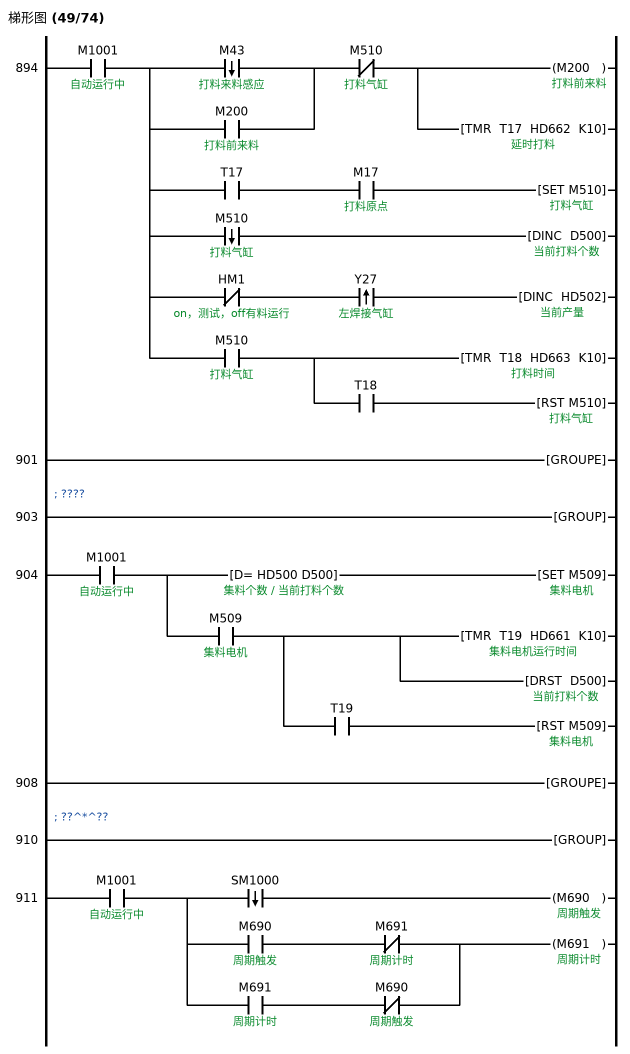
[picture p48: 梯形图 rows 894-911]
LD     M1001	; 自动运行中
MPS
LDF    M43	; 打料来料感应
OR     M200	; 打料前来料
ANB
ANI    M510	; 打料气缸
OUT    M200	; 打料前来料
TMR    T17 HD662 K10	; 延时打料
MRD
AND    T17
AND    M17	; 打料原点
SET    M510	; 打料气缸
MRD
ANDF   M510	; 打料气缸
DINC   D500	; 当前打料个数
MRD
ANI    HM1	; on，测试，off有料运行
ANDP   Y27	; 左焊接气缸
DINC   HD502	; 当前产量
MPP
AND    M510	; 打料气缸
TMR    T18 HD663 K10	; 打料时间
AND    T18
RST    M510	; 打料气缸
GROUPE
; ????
GROUP
LD     M1001	; 自动运行中
MPS
DAND=  HD500 D500	; 集料个数 / 当前打料个数
SET    M509	; 集料电机
MPP
AND    M509	; 集料电机
TMR    T19 HD661 K10	; 集料电机运行时间
DRST   D500	; 当前打料个数
AND    T19
RST    M509	; 集料电机
GROUPE
; ??^*^??
GROUP
LD     M1001	; 自动运行中
MPS
ANDF   SM1000
OUT    M690	; 周期触发
MPP
LD     M690	; 周期触发
ANI    M691	; 周期计时
LD     M691	; 周期计时
ANI    M690	; 周期触发
ORB
ANB
OUT    M691	; 周期计时

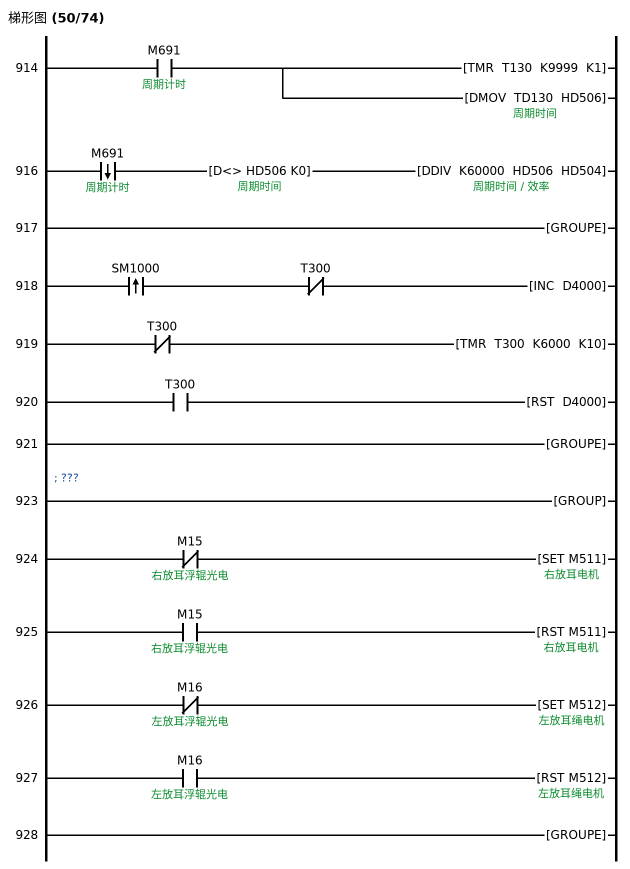
LD     M691	; 周期计时
TMR    T130 K9999 K1
DMOV   TD130 HD506	; 周期时间
LDF    M691	; 周期计时
DAND<> HD506 K0	; 周期时间
DDIV   K60000 HD506 HD504	; 周期时间 / 效率
GROUPE
LDP    SM1000
ANI    T300
INC    D4000
LDI    T300
TMR    T300 K6000 K10
LD     T300
RST    D4000
GROUPE
; ???
GROUP
LDI    M15	; 右放耳浮辊光电
SET    M511	; 右放耳电机
LD     M15	; 右放耳浮辊光电
RST    M511	; 右放耳电机
LDI    M16	; 左放耳浮辊光电
SET    M512	; 左放耳绳电机
LD     M16	; 左放耳浮辊光电
RST    M512	; 左放耳绳电机
GROUPE

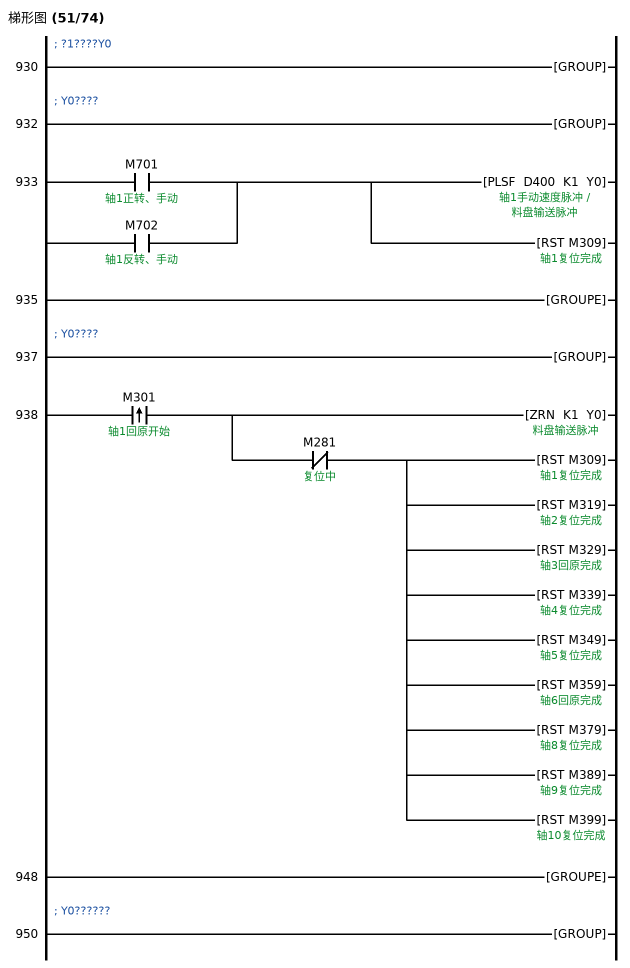
; ?1????Y0
GROUP
; Y0????
GROUP
LD     M701	; 轴1正转、手动
OR     M702	; 轴1反转、手动
PLSF   D400 K1 Y0	; 轴1手动速度脉冲 / 料盘输送脉冲
RST    M309	; 轴1复位完成
GROUPE
; Y0????
GROUP
LDP    M301	; 轴1回原开始
ZRN    K1 Y0	; 料盘输送脉冲
ANI    M281	; 复位中
RST    M309	; 轴1复位完成
RST    M319	; 轴2复位完成
RST    M329	; 轴3回原完成
RST    M339	; 轴4复位完成
RST    M349	; 轴5复位完成
RST    M359	; 轴6回原完成
RST    M379	; 轴8复位完成
RST    M389	; 轴9复位完成
RST    M399	; 轴10复位完成
GROUPE
; Y0??????
GROUP

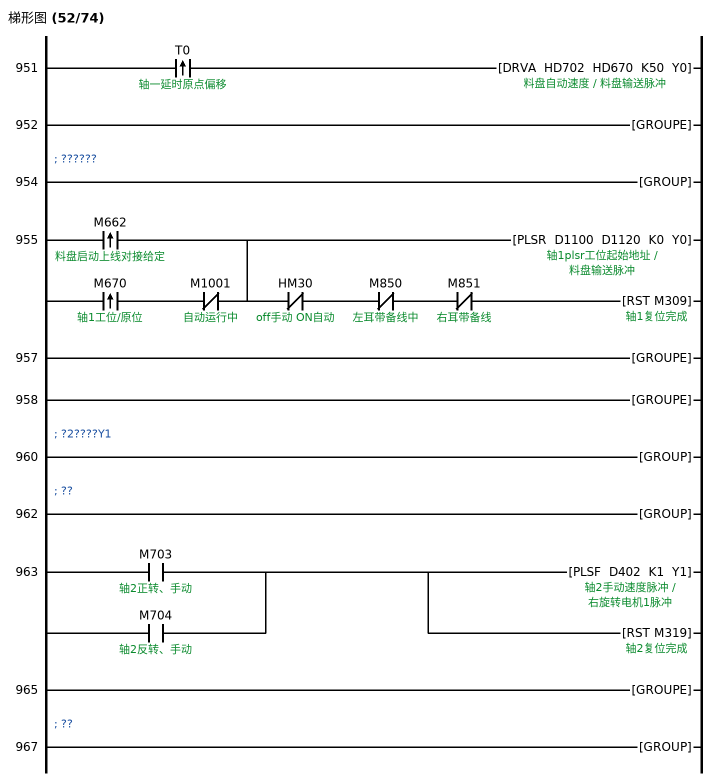
LDP    T0	; 轴一延时原点偏移
DRVA   HD702 HD670 K50 Y0	; 料盘自动速度 / 料盘输送脉冲
GROUPE
; ??????
GROUP
LDP    M662	; 料盘启动上线对接给定
LDP    M670	; 轴1工位/原位
ANI    M1001	; 自动运行中
ORB
PLSR   D1100 D1120 K0 Y0	; 轴1plsr工位起始地址 / 料盘输送脉冲
ANI    HM30	; off手动 ON自动
ANI    M850	; 左耳带备线中
ANI    M851	; 右耳带备线
RST    M309	; 轴1复位完成
GROUPE
GROUPE
; ?2????Y1
GROUP
; ??
GROUP
LD     M703	; 轴2正转、手动
OR     M704	; 轴2反转、手动
PLSF   D402 K1 Y1	; 轴2手动速度脉冲 / 右旋转电机1脉冲
RST    M319	; 轴2复位完成
GROUPE
; ??
GROUP

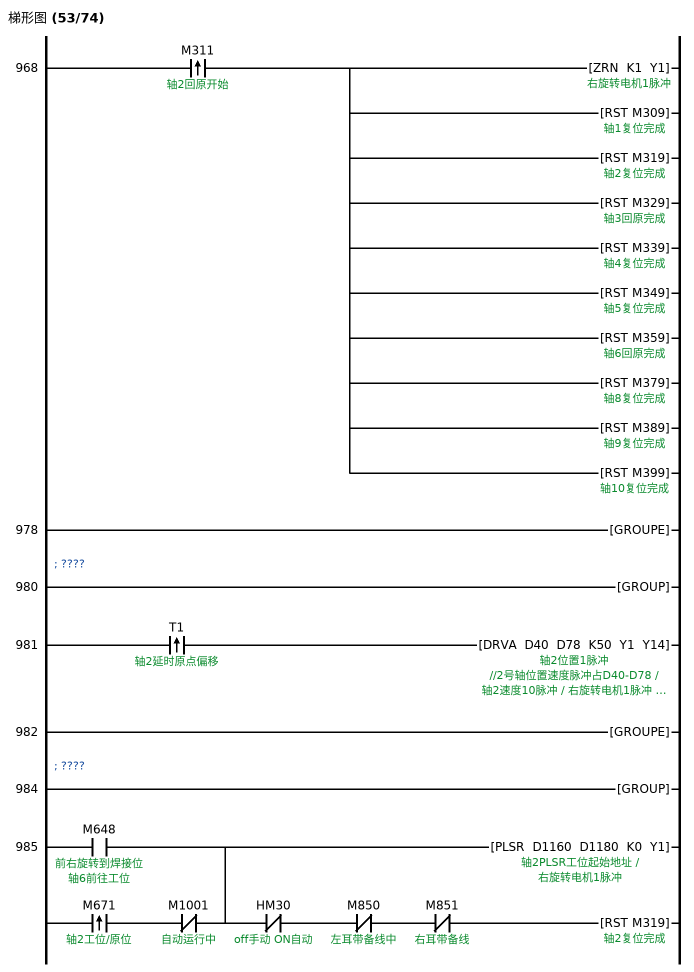
LDP    M311	; 轴2回原开始
ZRN    K1 Y1	; 右旋转电机1脉冲
RST    M309	; 轴1复位完成
RST    M319	; 轴2复位完成
RST    M329	; 轴3回原完成
RST    M339	; 轴4复位完成
RST    M349	; 轴5复位完成
RST    M359	; 轴6回原完成
RST    M379	; 轴8复位完成
RST    M389	; 轴9复位完成
RST    M399	; 轴10复位完成
GROUPE
; ????
GROUP
LDP    T1	; 轴2延时原点偏移
DRVA   D40 D78 K50 Y1 Y14	; 轴2位置1脉冲    //2号轴位置速度脉冲占D40-D78 / 轴2速度10脉冲 / 右旋转电机1脉冲 / 右旋转电机1方向
GROUPE
; ????
GROUP
LD     M648	; 前右旋转到焊接位 轴6前往工位
LDP    M671	; 轴2工位/原位
ANI    M1001	; 自动运行中
ORB
PLSR   D1160 D1180 K0 Y1	; 轴2PLSR工位起始地址 / 右旋转电机1脉冲
ANI    HM30	; off手动 ON自动
ANI    M850	; 左耳带备线中
ANI    M851	; 右耳带备线
RST    M319	; 轴2复位完成

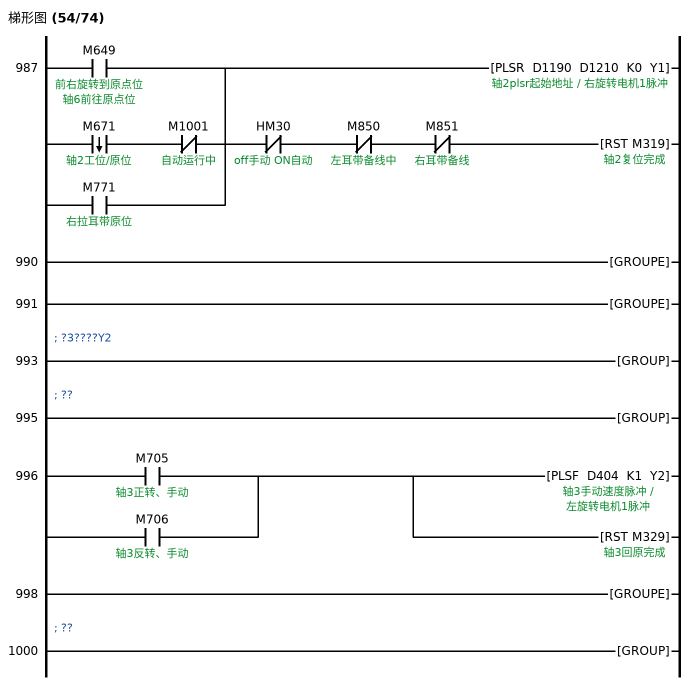
LD     M649	; 前右旋转到原点位 轴6前往原点位
LDF    M671	; 轴2工位/原位
ANI    M1001	; 自动运行中
ORB
OR     M771	; 右拉耳带原位
PLSR   D1190 D1210 K0 Y1	; 轴2plsr起始地址 / 右旋转电机1脉冲
ANI    HM30	; off手动 ON自动
ANI    M850	; 左耳带备线中
ANI    M851	; 右耳带备线
RST    M319	; 轴2复位完成
GROUPE
GROUPE
; ?3????Y2
GROUP
; ??
GROUP
LD     M705	; 轴3正转、手动
OR     M706	; 轴3反转、手动
PLSF   D404 K1 Y2	; 轴3手动速度脉冲 / 左旋转电机1脉冲
RST    M329	; 轴3回原完成
GROUPE
; ??
GROUP

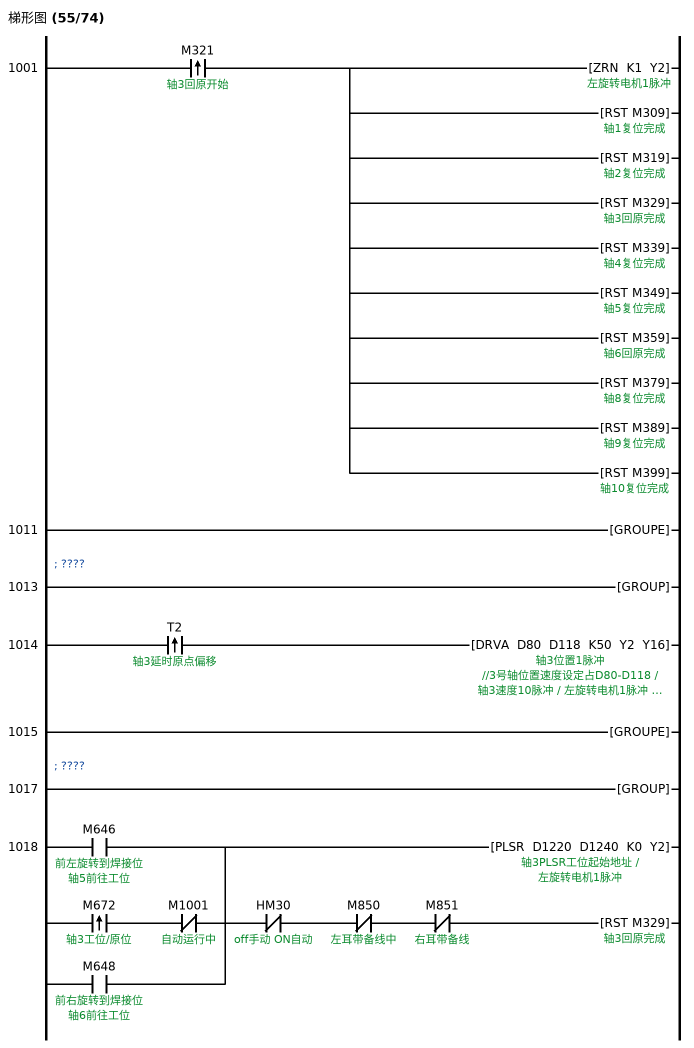
LDP    M321	; 轴3回原开始
ZRN    K1 Y2	; 左旋转电机1脉冲
RST    M309	; 轴1复位完成
RST    M319	; 轴2复位完成
RST    M329	; 轴3回原完成
RST    M339	; 轴4复位完成
RST    M349	; 轴5复位完成
RST    M359	; 轴6回原完成
RST    M379	; 轴8复位完成
RST    M389	; 轴9复位完成
RST    M399	; 轴10复位完成
GROUPE
; ????
GROUP
LDP    T2	; 轴3延时原点偏移
DRVA   D80 D118 K50 Y2 Y16	; 轴3位置1脉冲   //3号轴位置速度设定占D80-D118 / 轴3速度10脉冲 / 左旋转电机1脉冲 / 左旋转电机1方向
GROUPE
; ????
GROUP
LD     M646	; 前左旋转到焊接位 轴5前往工位
LDP    M672	; 轴3工位/原位
ANI    M1001	; 自动运行中
ORB
OR     M648	; 前右旋转到焊接位 轴6前往工位
PLSR   D1220 D1240 K0 Y2	; 轴3PLSR工位起始地址 / 左旋转电机1脉冲
ANI    HM30	; off手动 ON自动
ANI    M850	; 左耳带备线中
ANI    M851	; 右耳带备线
RST    M329	; 轴3回原完成

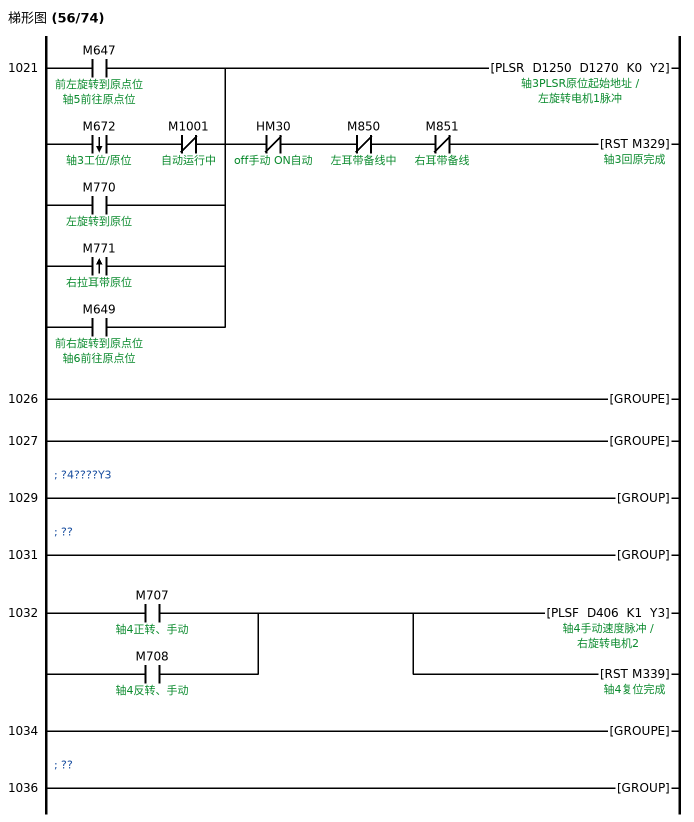
LD     M647	; 前左旋转到原点位 轴5前往原点位
LDF    M672	; 轴3工位/原位
ANI    M1001	; 自动运行中
ORB
OR     M770	; 左旋转到原位
ORP    M771	; 右拉耳带原位
OR     M649	; 前右旋转到原点位 轴6前往原点位
PLSR   D1250 D1270 K0 Y2	; 轴3PLSR原位起始地址 / 左旋转电机1脉冲
ANI    HM30	; off手动 ON自动
ANI    M850	; 左耳带备线中
ANI    M851	; 右耳带备线
RST    M329	; 轴3回原完成
GROUPE
GROUPE
; ?4????Y3
GROUP
; ??
GROUP
LD     M707	; 轴4正转、手动
OR     M708	; 轴4反转、手动
PLSF   D406 K1 Y3	; 轴4手动速度脉冲 / 右旋转电机2
RST    M339	; 轴4复位完成
GROUPE
; ??
GROUP

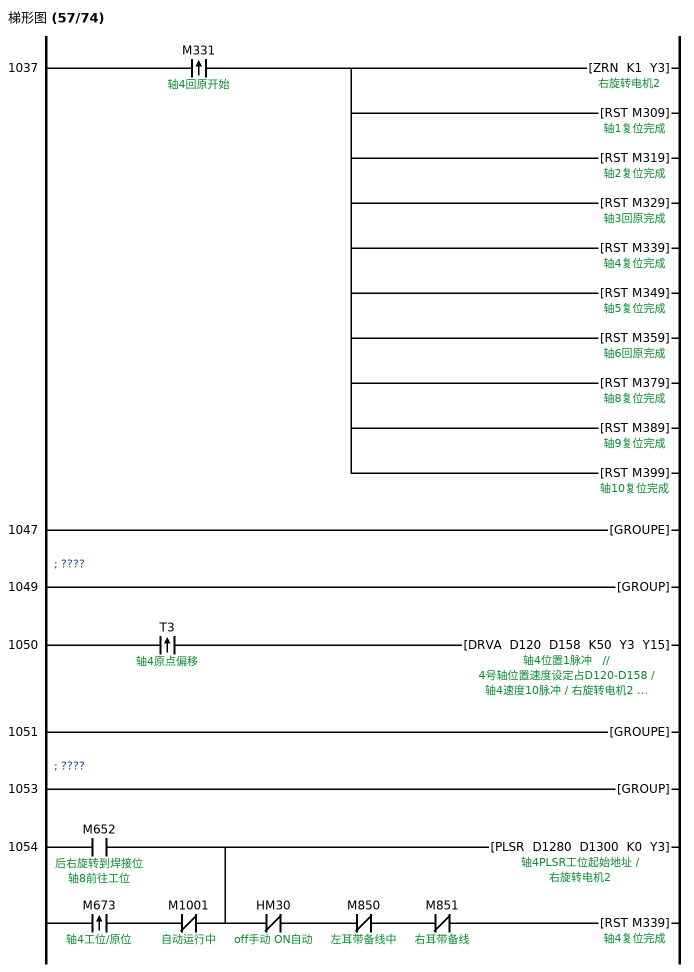
LDP    M331	; 轴4回原开始
ZRN    K1 Y3	; 右旋转电机2
RST    M309	; 轴1复位完成
RST    M319	; 轴2复位完成
RST    M329	; 轴3回原完成
RST    M339	; 轴4复位完成
RST    M349	; 轴5复位完成
RST    M359	; 轴6回原完成
RST    M379	; 轴8复位完成
RST    M389	; 轴9复位完成
RST    M399	; 轴10复位完成
GROUPE
; ????
GROUP
LDP    T3	; 轴4原点偏移
DRVA   D120 D158 K50 Y3 Y15	; 轴4位置1脉冲   //4号轴位置速度设定占D120-D158 / 轴4速度10脉冲 / 右旋转电机2 / 右旋转电机2方向
GROUPE
; ????
GROUP
LD     M652	; 后右旋转到焊接位 轴8前往工位
LDP    M673	; 轴4工位/原位
ANI    M1001	; 自动运行中
ORB
PLSR   D1280 D1300 K0 Y3	; 轴4PLSR工位起始地址 / 右旋转电机2
ANI    HM30	; off手动 ON自动
ANI    M850	; 左耳带备线中
ANI    M851	; 右耳带备线
RST    M339	; 轴4复位完成

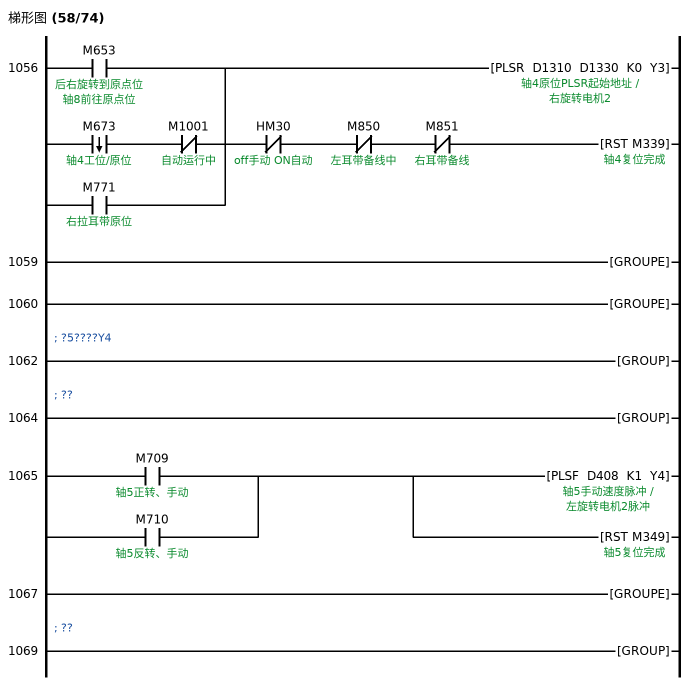
LD     M653	; 后右旋转到原点位 轴8前往原点位
LDF    M673	; 轴4工位/原位
ANI    M1001	; 自动运行中
ORB
OR     M771	; 右拉耳带原位
PLSR   D1310 D1330 K0 Y3	; 轴4原位PLSR起始地址 / 右旋转电机2
ANI    HM30	; off手动 ON自动
ANI    M850	; 左耳带备线中
ANI    M851	; 右耳带备线
RST    M339	; 轴4复位完成
GROUPE
GROUPE
; ?5????Y4
GROUP
; ??
GROUP
LD     M709	; 轴5正转、手动
OR     M710	; 轴5反转、手动
PLSF   D408 K1 Y4	; 轴5手动速度脉冲 / 左旋转电机2脉冲
RST    M349	; 轴5复位完成
GROUPE
; ??
GROUP

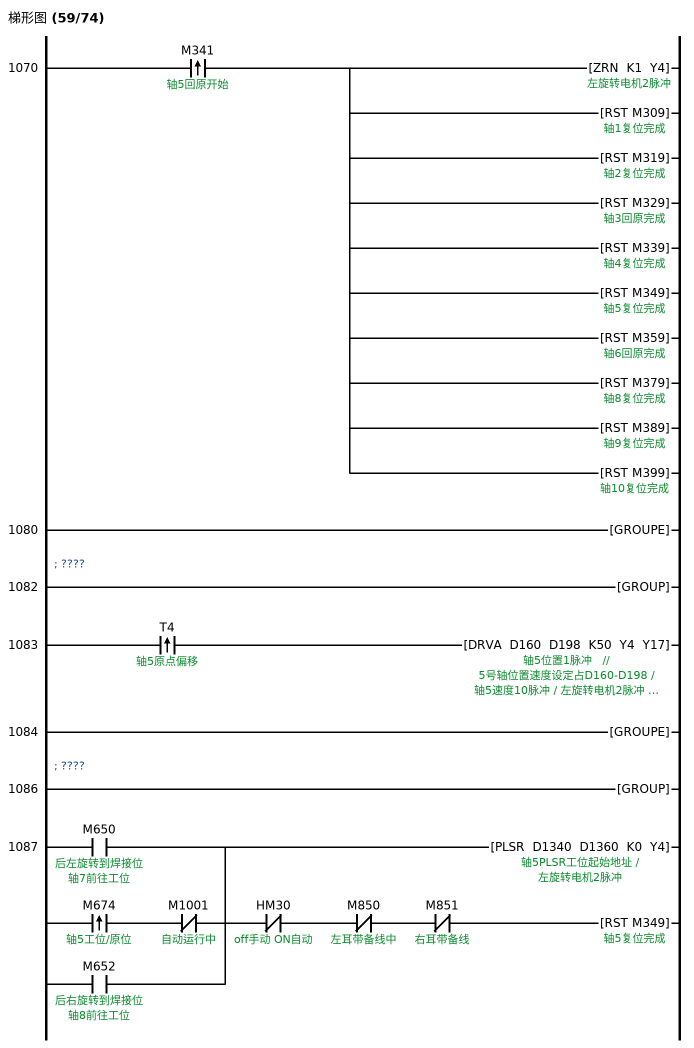
LDP    M341	; 轴5回原开始
ZRN    K1 Y4	; 左旋转电机2脉冲
RST    M309	; 轴1复位完成
RST    M319	; 轴2复位完成
RST    M329	; 轴3回原完成
RST    M339	; 轴4复位完成
RST    M349	; 轴5复位完成
RST    M359	; 轴6回原完成
RST    M379	; 轴8复位完成
RST    M389	; 轴9复位完成
RST    M399	; 轴10复位完成
GROUPE
; ????
GROUP
LDP    T4	; 轴5原点偏移
DRVA   D160 D198 K50 Y4 Y17	; 轴5位置1脉冲   //5号轴位置速度设定占D160-D198 / 轴5速度10脉冲 / 左旋转电机2脉冲 / 左旋转电机2方向
GROUPE
; ????
GROUP
LD     M650	; 后左旋转到焊接位 轴7前往工位
LDP    M674	; 轴5工位/原位
ANI    M1001	; 自动运行中
ORB
OR     M652	; 后右旋转到焊接位 轴8前往工位
PLSR   D1340 D1360 K0 Y4	; 轴5PLSR工位起始地址 / 左旋转电机2脉冲
ANI    HM30	; off手动 ON自动
ANI    M850	; 左耳带备线中
ANI    M851	; 右耳带备线
RST    M349	; 轴5复位完成

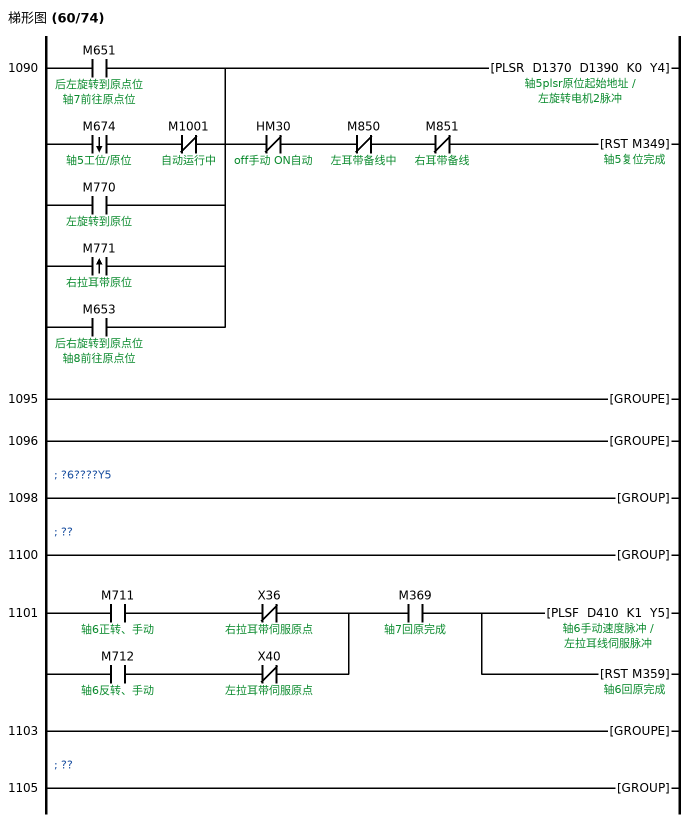
LD     M651	; 后左旋转到原点位 轴7前往原点位
LDF    M674	; 轴5工位/原位
ANI    M1001	; 自动运行中
ORB
OR     M770	; 左旋转到原位
ORP    M771	; 右拉耳带原位
OR     M653	; 后右旋转到原点位 轴8前往原点位
PLSR   D1370 D1390 K0 Y4	; 轴5plsr原位起始地址 / 左旋转电机2脉冲
ANI    HM30	; off手动 ON自动
ANI    M850	; 左耳带备线中
ANI    M851	; 右耳带备线
RST    M349	; 轴5复位完成
GROUPE
GROUPE
; ?6????Y5
GROUP
; ??
GROUP
LD     M711	; 轴6正转、手动
ANI    X36	; 右拉耳带伺服原点
LD     M712	; 轴6反转、手动
ANI    X40	; 左拉耳带伺服原点
ORB
AND    M369	; 轴7回原完成
PLSF   D410 K1 Y5	; 轴6手动速度脉冲 / 左拉耳线伺服脉冲
RST    M359	; 轴6回原完成
GROUPE
; ??
GROUP

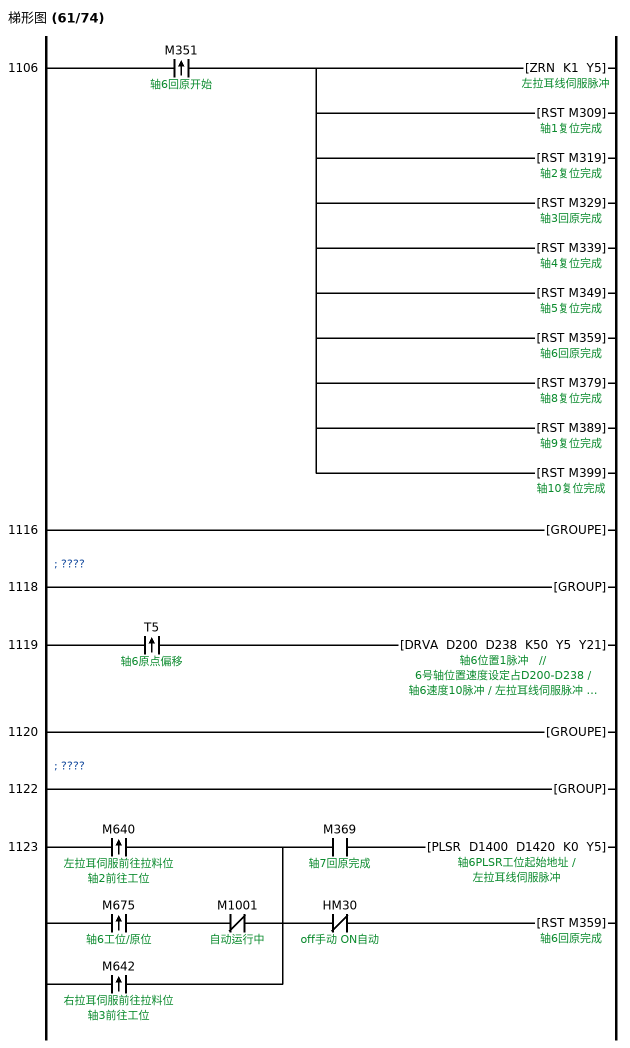
LDP    M351	; 轴6回原开始
ZRN    K1 Y5	; 左拉耳线伺服脉冲
RST    M309	; 轴1复位完成
RST    M319	; 轴2复位完成
RST    M329	; 轴3回原完成
RST    M339	; 轴4复位完成
RST    M349	; 轴5复位完成
RST    M359	; 轴6回原完成
RST    M379	; 轴8复位完成
RST    M389	; 轴9复位完成
RST    M399	; 轴10复位完成
GROUPE
; ????
GROUP
LDP    T5	; 轴6原点偏移
DRVA   D200 D238 K50 Y5 Y21	; 轴6位置1脉冲   //6号轴位置速度设定占D200-D238 / 轴6速度10脉冲 / 左拉耳线伺服脉冲 / 左拉耳带伺服方向
GROUPE
; ????
GROUP
LDP    M640	; 左拉耳伺服前往拉料位 轴2前往工位
LDP    M675	; 轴6工位/原位
ANI    M1001	; 自动运行中
ORB
ORP    M642	; 右拉耳伺服前往拉料位 轴3前往工位
MPS
AND    M369	; 轴7回原完成
PLSR   D1400 D1420 K0 Y5	; 轴6PLSR工位起始地址 / 左拉耳线伺服脉冲
MPP
ANI    HM30	; off手动 ON自动
RST    M359	; 轴6回原完成

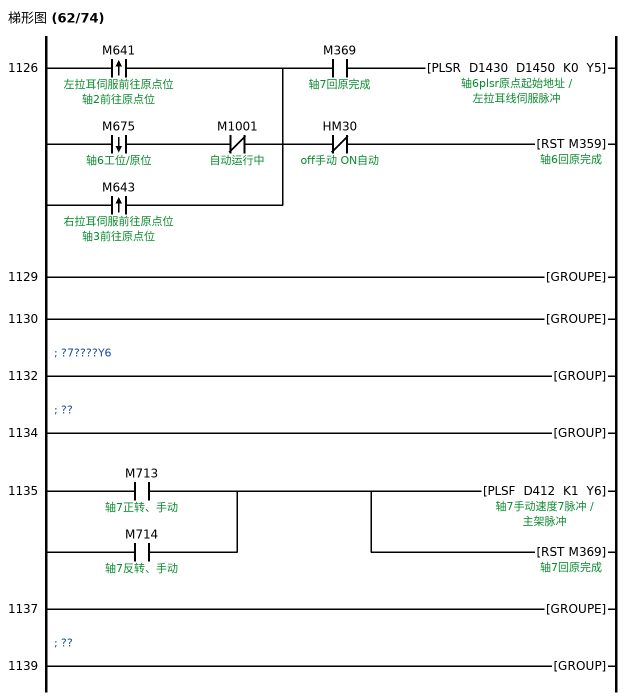
LDP    M641	; 左拉耳伺服前往原点位 轴2前往原点位
LDF    M675	; 轴6工位/原位
ANI    M1001	; 自动运行中
ORB
ORP    M643	; 右拉耳伺服前往原点位 轴3前往原点位
MPS
AND    M369	; 轴7回原完成
PLSR   D1430 D1450 K0 Y5	; 轴6plsr原点起始地址 / 左拉耳线伺服脉冲
MPP
ANI    HM30	; off手动 ON自动
RST    M359	; 轴6回原完成
GROUPE
GROUPE
; ?7????Y6
GROUP
; ??
GROUP
LD     M713	; 轴7正转、手动
OR     M714	; 轴7反转、手动
PLSF   D412 K1 Y6	; 轴7手动速度7脉冲 / 主架脉冲
RST    M369	; 轴7回原完成
GROUPE
; ??
GROUP

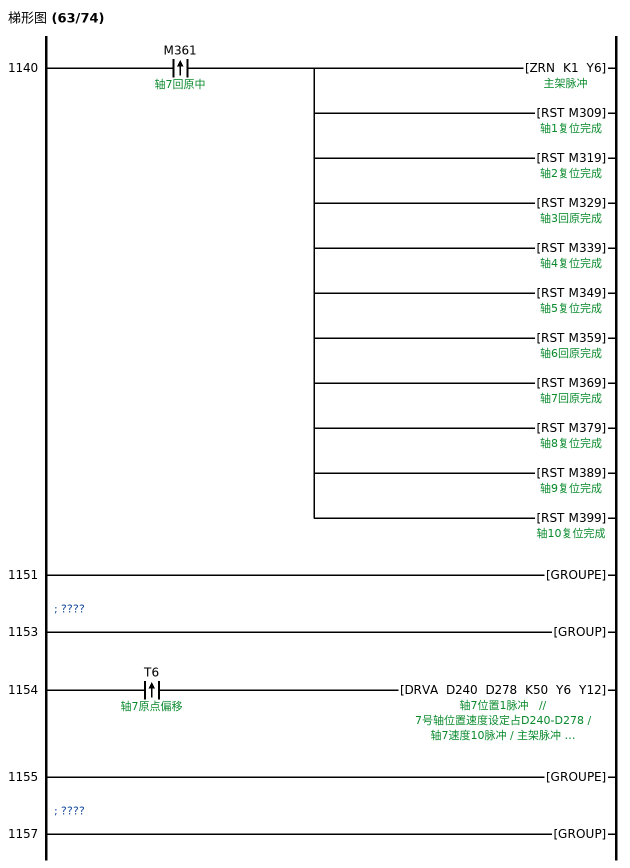
LDP    M361	; 轴7回原中
ZRN    K1 Y6	; 主架脉冲
RST    M309	; 轴1复位完成
RST    M319	; 轴2复位完成
RST    M329	; 轴3回原完成
RST    M339	; 轴4复位完成
RST    M349	; 轴5复位完成
RST    M359	; 轴6回原完成
RST    M369	; 轴7回原完成
RST    M379	; 轴8复位完成
RST    M389	; 轴9复位完成
RST    M399	; 轴10复位完成
GROUPE
; ????
GROUP
LDP    T6	; 轴7原点偏移
DRVA   D240 D278 K50 Y6 Y12	; 轴7位置1脉冲   //7号轴位置速度设定占D240-D278 / 轴7速度10脉冲 / 主架脉冲 / 主架伺服方向
GROUPE
; ????
GROUP

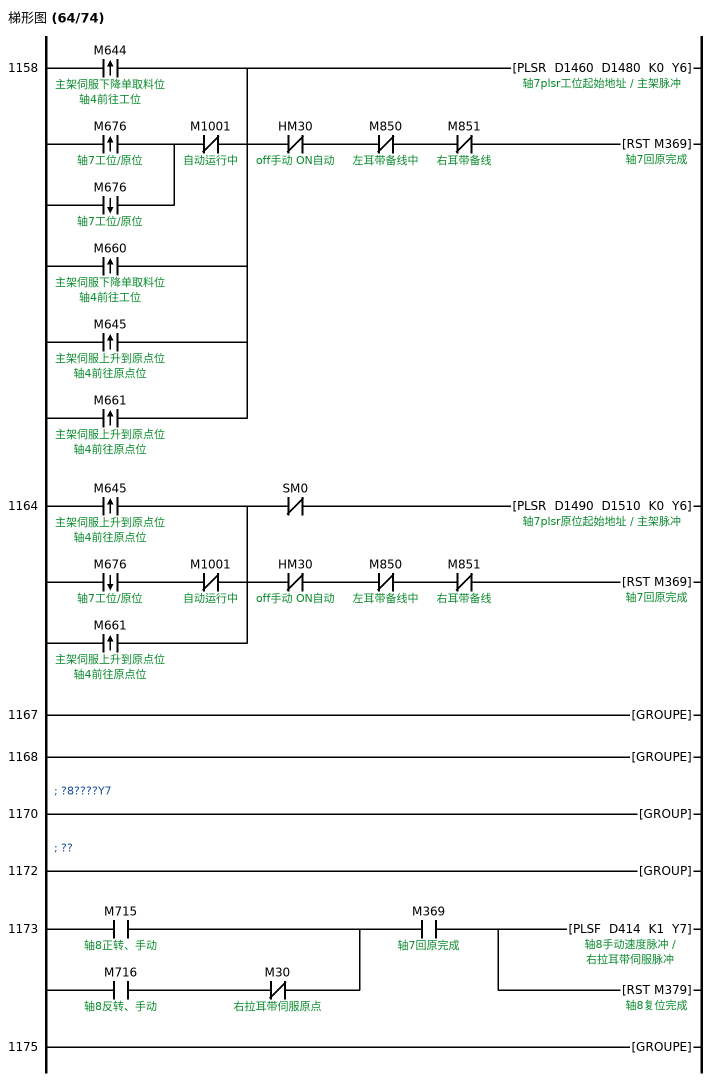
LDP    M644	; 主架伺服下降单取料位 轴4前往工位
LDP    M676	; 轴7工位/原位
ORF    M676	; 轴7工位/原位
ANI    M1001	; 自动运行中
ORB
ORP    M660	; 主架伺服下降单取料位 轴4前往工位
ORP    M645	; 主架伺服上升到原点位 轴4前往原点位
ORP    M661	; 主架伺服上升到原点位 轴4前往原点位
PLSR   D1460 D1480 K0 Y6	; 轴7plsr工位起始地址 / 主架脉冲
ANI    HM30	; off手动 ON自动
ANI    M850	; 左耳带备线中
ANI    M851	; 右耳带备线
RST    M369	; 轴7回原完成
LDP    M645	; 主架伺服上升到原点位 轴4前往原点位
LDF    M676	; 轴7工位/原位
ANI    M1001	; 自动运行中
ORB
ORP    M661	; 主架伺服上升到原点位 轴4前往原点位
MPS
ANI    SM0
PLSR   D1490 D1510 K0 Y6	; 轴7plsr原位起始地址 / 主架脉冲
MPP
ANI    HM30	; off手动 ON自动
ANI    M850	; 左耳带备线中
ANI    M851	; 右耳带备线
RST    M369	; 轴7回原完成
GROUPE
GROUPE
; ?8????Y7
GROUP
; ??
GROUP
LD     M715	; 轴8正转、手动
LD     M716	; 轴8反转、手动
ANI    M30	; 右拉耳带伺服原点
ORB
AND    M369	; 轴7回原完成
PLSF   D414 K1 Y7	; 轴8手动速度脉冲 / 右拉耳带伺服脉冲
RST    M379	; 轴8复位完成
GROUPE

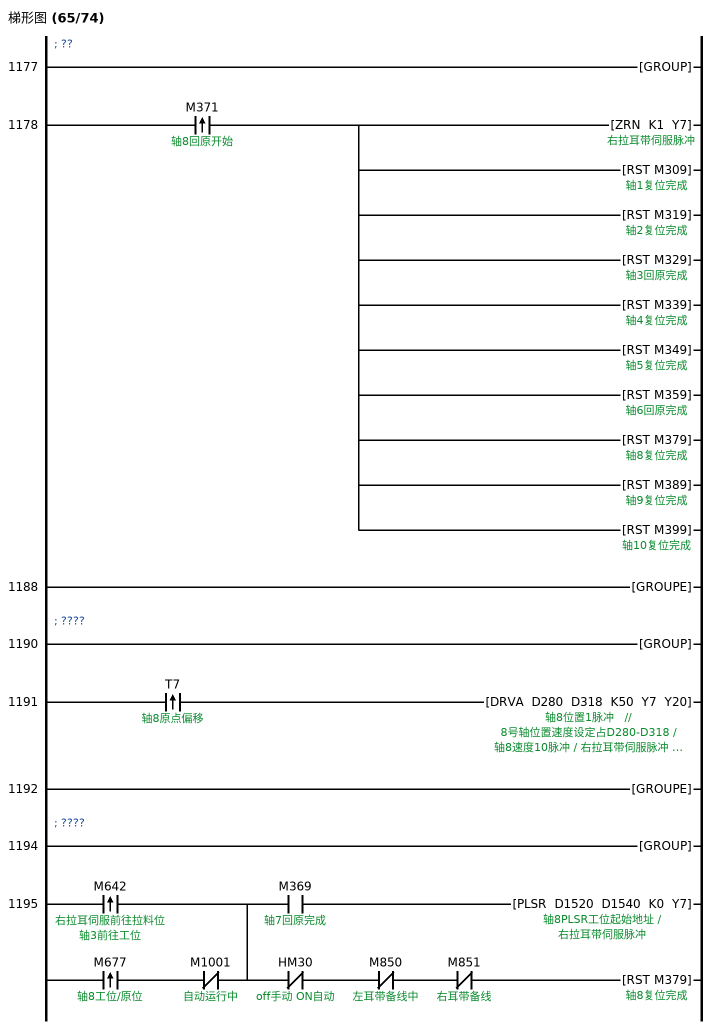
; ??
GROUP
LDP    M371	; 轴8回原开始
ZRN    K1 Y7	; 右拉耳带伺服脉冲
RST    M309	; 轴1复位完成
RST    M319	; 轴2复位完成
RST    M329	; 轴3回原完成
RST    M339	; 轴4复位完成
RST    M349	; 轴5复位完成
RST    M359	; 轴6回原完成
RST    M379	; 轴8复位完成
RST    M389	; 轴9复位完成
RST    M399	; 轴10复位完成
GROUPE
; ????
GROUP
LDP    T7	; 轴8原点偏移
DRVA   D280 D318 K50 Y7 Y20	; 轴8位置1脉冲   //8号轴位置速度设定占D280-D318 / 轴8速度10脉冲 / 右拉耳带伺服脉冲 / 右拉耳带伺服方向
GROUPE
; ????
GROUP
LDP    M642	; 右拉耳伺服前往拉料位 轴3前往工位
LDP    M677	; 轴8工位/原位
ANI    M1001	; 自动运行中
ORB
MPS
AND    M369	; 轴7回原完成
PLSR   D1520 D1540 K0 Y7	; 轴8PLSR工位起始地址 / 右拉耳带伺服脉冲
MPP
ANI    HM30	; off手动 ON自动
ANI    M850	; 左耳带备线中
ANI    M851	; 右耳带备线
RST    M379	; 轴8复位完成

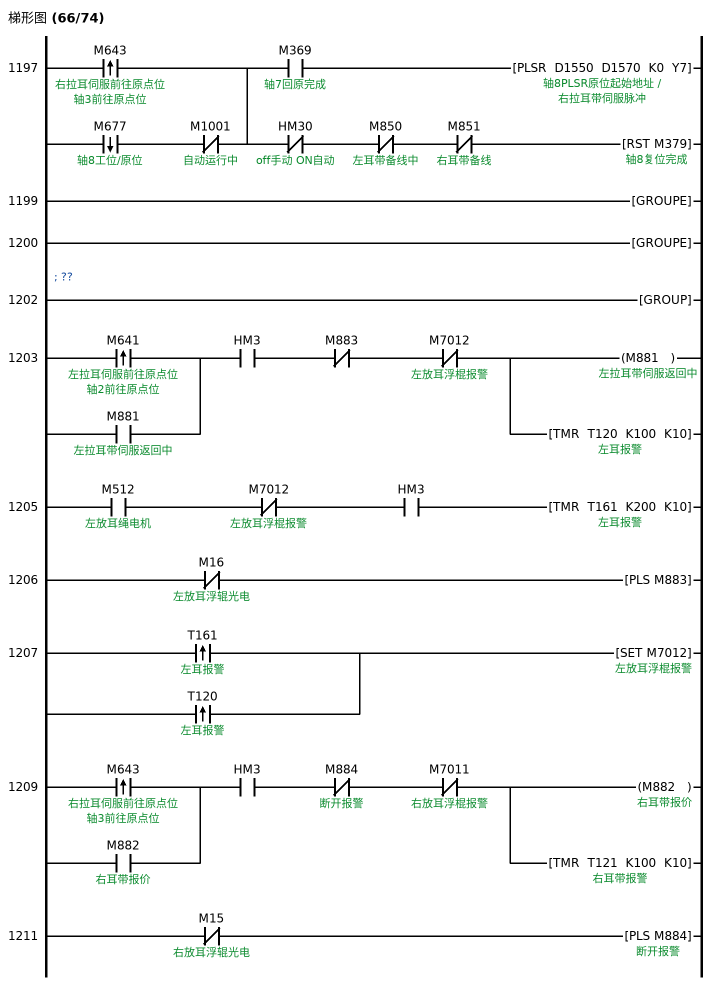
LDP    M643	; 右拉耳伺服前往原点位 轴3前往原点位
LDF    M677	; 轴8工位/原位
ANI    M1001	; 自动运行中
ORB
MPS
AND    M369	; 轴7回原完成
PLSR   D1550 D1570 K0 Y7	; 轴8PLSR原位起始地址 / 右拉耳带伺服脉冲
MPP
ANI    HM30	; off手动 ON自动
ANI    M850	; 左耳带备线中
ANI    M851	; 右耳带备线
RST    M379	; 轴8复位完成
GROUPE
GROUPE
; ??
GROUP
LDP    M641	; 左拉耳伺服前往原点位 轴2前往原点位
OR     M881	; 左拉耳带伺服返回中
AND    HM3
ANI    M883
ANI    M7012	; 左放耳浮棍报警
OUT    M881	; 左拉耳带伺服返回中
TMR    T120 K100 K10	; 左耳报警
LD     M512	; 左放耳绳电机
ANI    M7012	; 左放耳浮棍报警
AND    HM3
TMR    T161 K200 K10	; 左耳报警
LDI    M16	; 左放耳浮辊光电
PLS    M883
LDP    T161	; 左耳报警
ORP    T120	; 左耳报警
SET    M7012	; 左放耳浮棍报警
LDP    M643	; 右拉耳伺服前往原点位 轴3前往原点位
OR     M882	; 右耳带报价
AND    HM3
ANI    M884	; 断开报警
ANI    M7011	; 右放耳浮棍报警
OUT    M882	; 右耳带报价
TMR    T121 K100 K10	; 右耳带报警
LDI    M15	; 右放耳浮辊光电
PLS    M884	; 断开报警

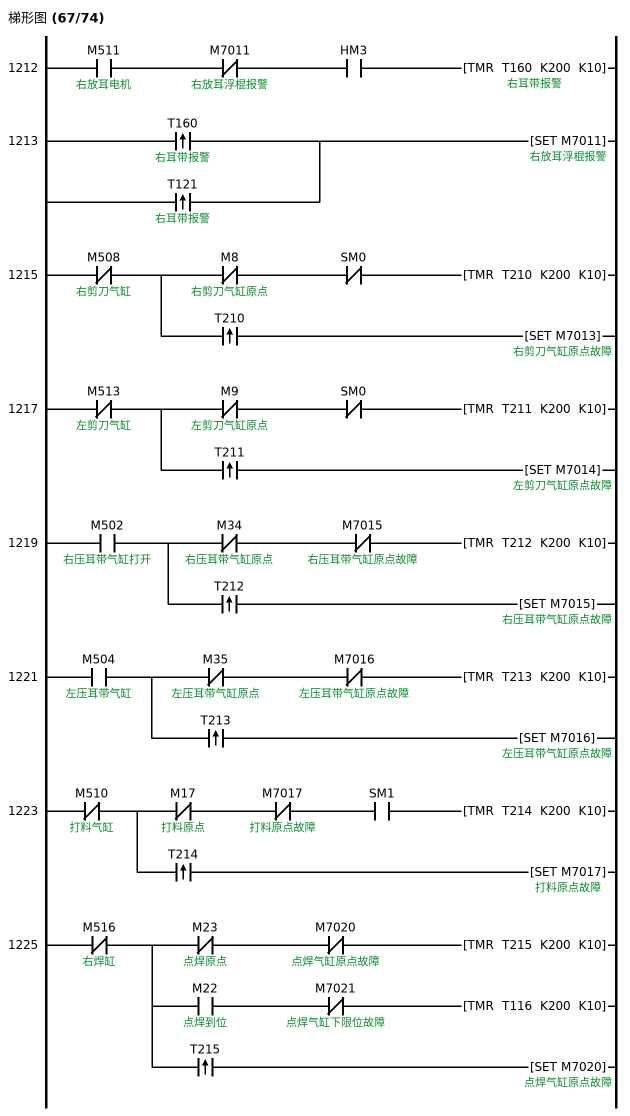
LD     M511	; 右放耳电机
ANI    M7011	; 右放耳浮棍报警
AND    HM3
TMR    T160 K200 K10	; 右耳带报警
LDP    T160	; 右耳带报警
ORP    T121	; 右耳带报警
SET    M7011	; 右放耳浮棍报警
LDI    M508	; 右剪刀气缸
MPS
ANI    M8	; 右剪刀气缸原点
ANI    SM0
TMR    T210 K200 K10
MPP
ANDP   T210
SET    M7013	; 右剪刀气缸原点故障
LDI    M513	; 左剪刀气缸
MPS
ANI    M9	; 左剪刀气缸原点
ANI    SM0
TMR    T211 K200 K10
MPP
ANDP   T211
SET    M7014	; 左剪刀气缸原点故障
LD     M502	; 右压耳带气缸打开
MPS
ANI    M34	; 右压耳带气缸原点
ANI    M7015	; 右压耳带气缸原点故障
TMR    T212 K200 K10
MPP
ANDP   T212
SET    M7015	; 右压耳带气缸原点故障
LD     M504	; 左压耳带气缸
MPS
ANI    M35	; 左压耳带气缸原点
ANI    M7016	; 左压耳带气缸原点故障
TMR    T213 K200 K10
MPP
ANDP   T213
SET    M7016	; 左压耳带气缸原点故障
LDI    M510	; 打料气缸
MPS
ANI    M17	; 打料原点
ANI    M7017	; 打料原点故障
AND    SM1
TMR    T214 K200 K10
MPP
ANDP   T214
SET    M7017	; 打料原点故障
LDI    M516	; 右焊缸
MPS
ANI    M23	; 点焊原点
ANI    M7020	; 点焊气缸原点故障
TMR    T215 K200 K10
MRD
AND    M22	; 点焊到位
ANI    M7021	; 点焊气缸下限位故障
TMR    T116 K200 K10
MPP
ANDP   T215
SET    M7020	; 点焊气缸原点故障

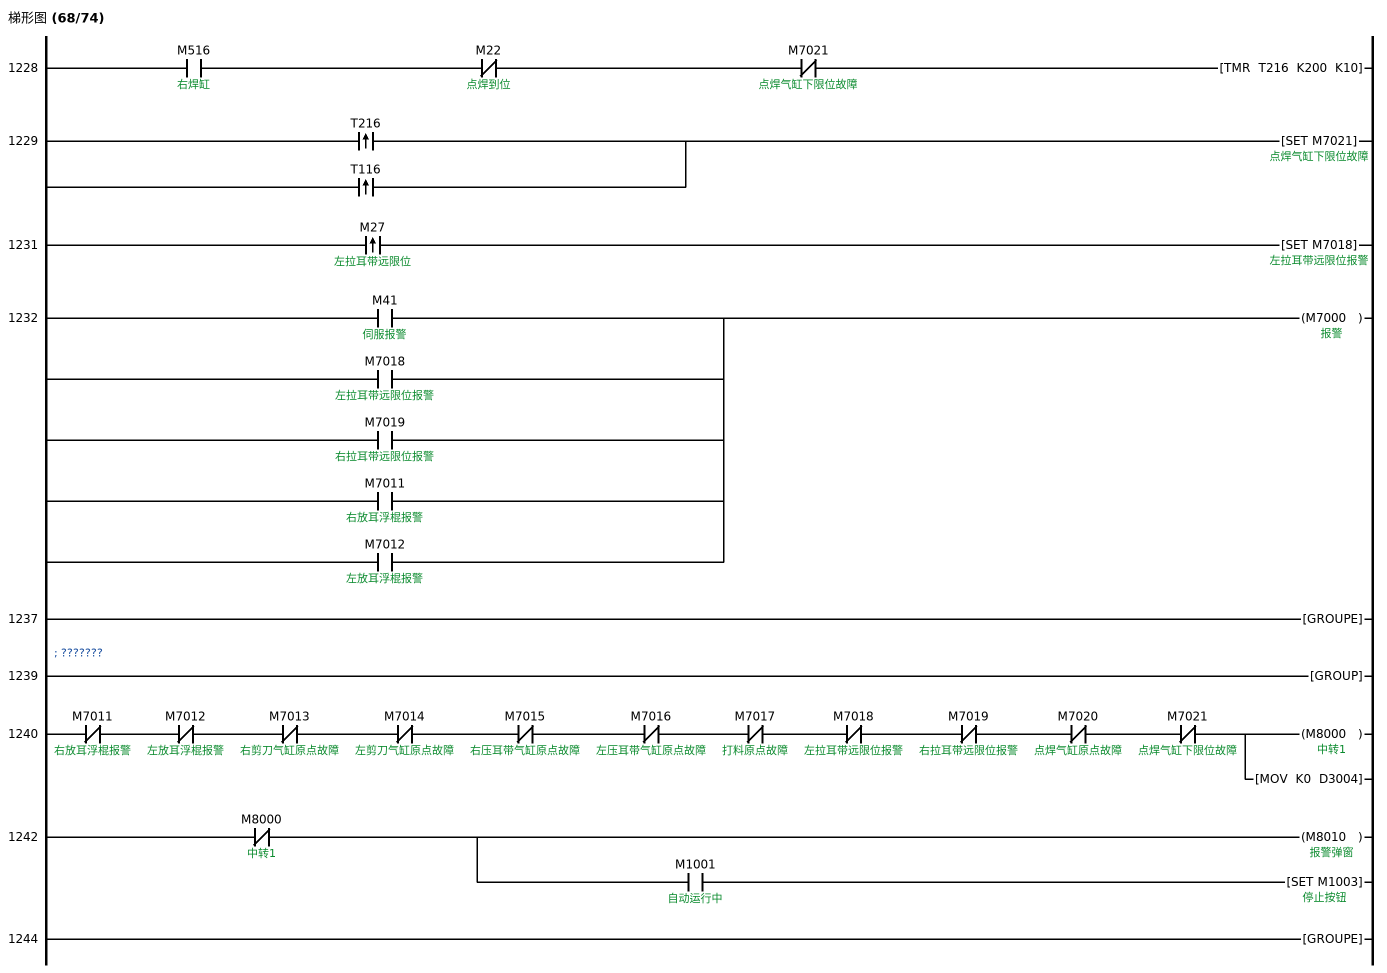
LD     M516	; 右焊缸
ANI    M22	; 点焊到位
ANI    M7021	; 点焊气缸下限位故障
TMR    T216 K200 K10
LDP    T216
ORP    T116
SET    M7021	; 点焊气缸下限位故障
LDP    M27	; 左拉耳带远限位
SET    M7018	; 左拉耳带远限位报警
LD     M41	; 伺服报警
OR     M7018	; 左拉耳带远限位报警
OR     M7019	; 右拉耳带远限位报警
OR     M7011	; 右放耳浮棍报警
OR     M7012	; 左放耳浮棍报警
OUT    M7000	; 报警
GROUPE
; ???????
GROUP
LDI    M7011	; 右放耳浮棍报警
ANI    M7012	; 左放耳浮棍报警
ANI    M7013	; 右剪刀气缸原点故障
ANI    M7014	; 左剪刀气缸原点故障
ANI    M7015	; 右压耳带气缸原点故障
ANI    M7016	; 左压耳带气缸原点故障
ANI    M7017	; 打料原点故障
ANI    M7018	; 左拉耳带远限位报警
ANI    M7019	; 右拉耳带远限位报警
ANI    M7020	; 点焊气缸原点故障
ANI    M7021	; 点焊气缸下限位故障
OUT    M8000	; 中转1
MOV    K0 D3004
LDI    M8000	; 中转1
OUT    M8010	; 报警弹窗
AND    M1001	; 自动运行中
SET    M1003	; 停止按钮
GROUPE

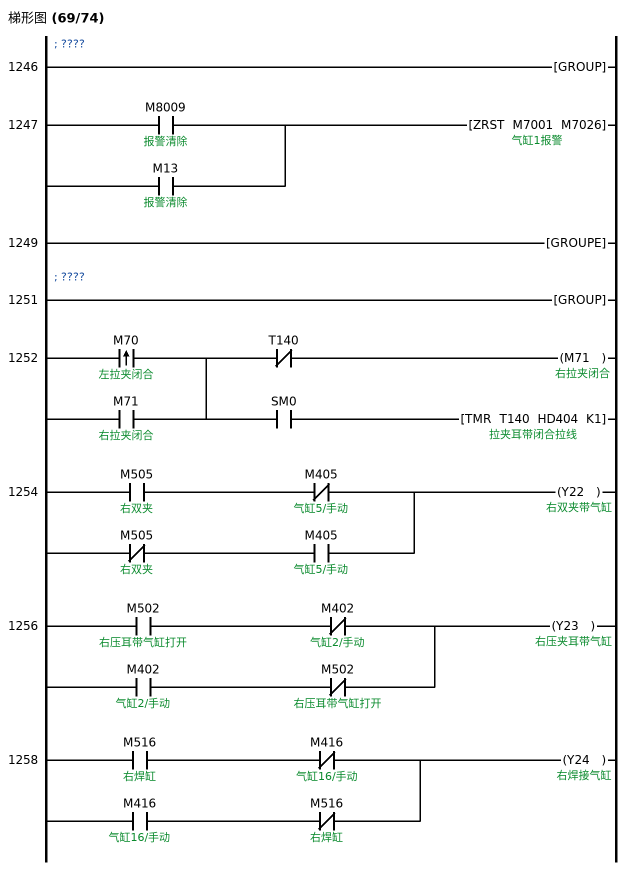
; ????
GROUP
LD     M8009	; 报警清除
OR     M13	; 报警清除
ZRST   M7001 M7026	; 气缸1报警
GROUPE
; ????
GROUP
LDP    M70	; 左拉夹闭合
OR     M71	; 右拉夹闭合
MPS
ANI    T140
OUT    M71	; 右拉夹闭合
MPP
AND    SM0
TMR    T140 HD404 K1	; 拉夹耳带闭合拉线
LD     M505	; 右双夹
ANI    M405	; 气缸5/手动
LDI    M505	; 右双夹
AND    M405	; 气缸5/手动
ORB
OUT    Y22	; 右双夹带气缸
LD     M502	; 右压耳带气缸打开
ANI    M402	; 气缸2/手动
LD     M402	; 气缸2/手动
ANI    M502	; 右压耳带气缸打开
ORB
OUT    Y23	; 右压夹耳带气缸
LD     M516	; 右焊缸
ANI    M416	; 气缸16/手动
LD     M416	; 气缸16/手动
ANI    M516	; 右焊缸
ORB
OUT    Y24	; 右焊接气缸

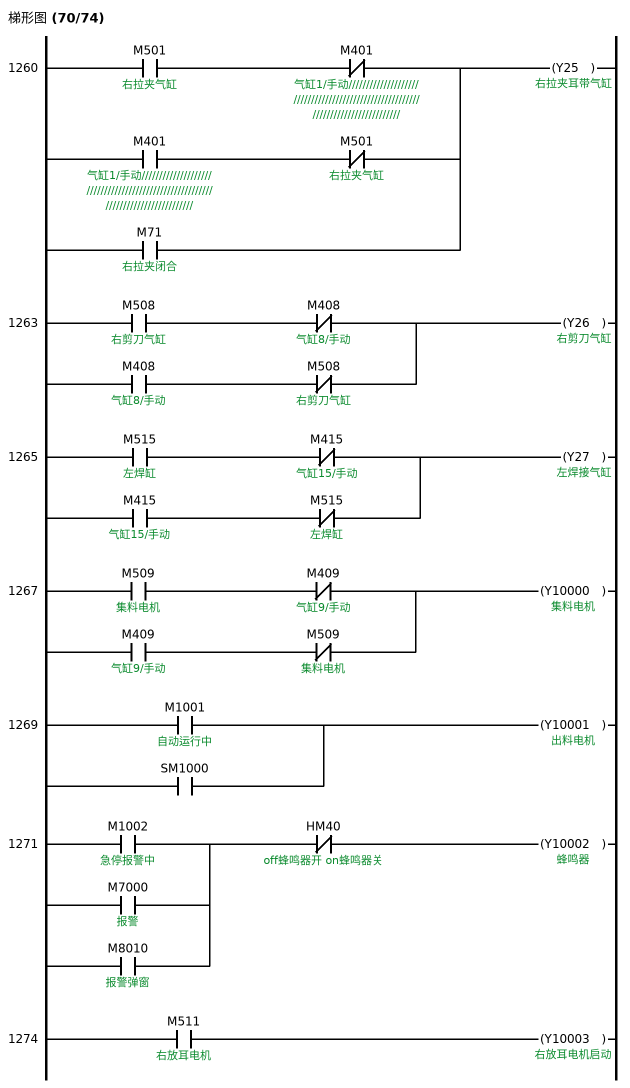
LD     M501	; 右拉夹气缸
ANI    M401	; 气缸1/手动/////////////////////////////////////////////////////////////////////////////////
LD     M401	; 气缸1/手动/////////////////////////////////////////////////////////////////////////////////
ANI    M501	; 右拉夹气缸
ORB
OR     M71	; 右拉夹闭合
OUT    Y25	; 右拉夹耳带气缸
LD     M508	; 右剪刀气缸
ANI    M408	; 气缸8/手动
LD     M408	; 气缸8/手动
ANI    M508	; 右剪刀气缸
ORB
OUT    Y26	; 右剪刀气缸
LD     M515	; 左焊缸
ANI    M415	; 气缸15/手动
LD     M415	; 气缸15/手动
ANI    M515	; 左焊缸
ORB
OUT    Y27	; 左焊接气缸
LD     M509	; 集料电机
ANI    M409	; 气缸9/手动
LD     M409	; 气缸9/手动
ANI    M509	; 集料电机
ORB
OUT    Y10000	; 集料电机
LD     M1001	; 自动运行中
OR     SM1000
OUT    Y10001	; 出料电机
LD     M1002	; 急停报警中
OR     M7000	; 报警
OR     M8010	; 报警弹窗
ANI    HM40	; off蜂鸣器开 on蜂鸣器关
OUT    Y10002	; 蜂鸣器
LD     M511	; 右放耳电机
OUT    Y10003	; 右放耳电机启动

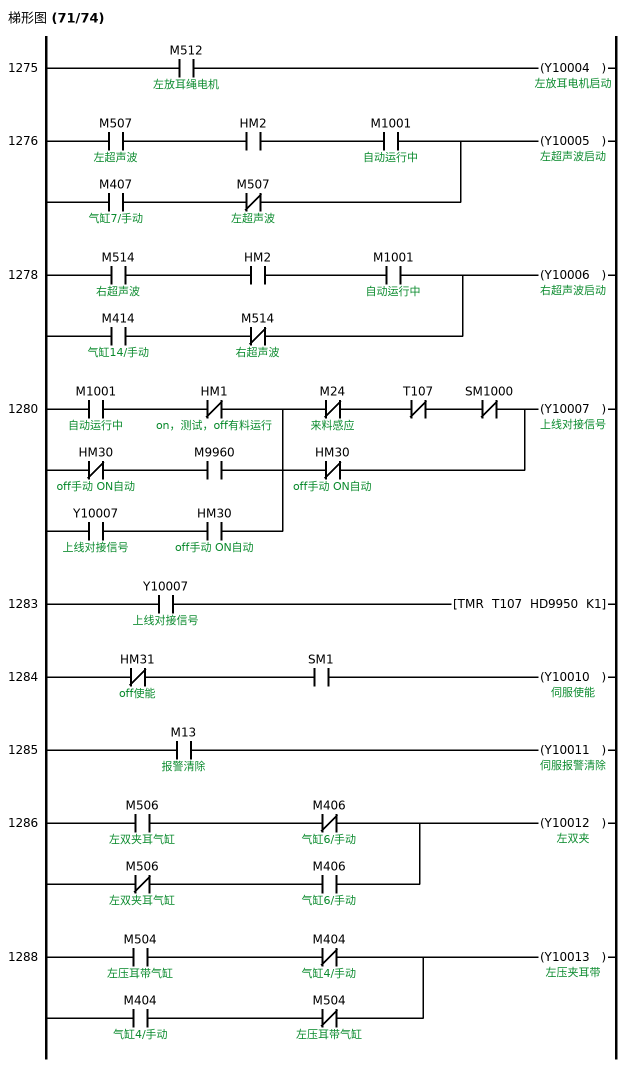
LD     M512	; 左放耳绳电机
OUT    Y10004	; 左放耳电机启动
LD     M507	; 左超声波
AND    HM2
AND    M1001	; 自动运行中
LD     M407	; 气缸7/手动
ANI    M507	; 左超声波
ORB
OUT    Y10005	; 左超声波启动
LD     M514	; 右超声波
AND    HM2
AND    M1001	; 自动运行中
LD     M414	; 气缸14/手动
ANI    M514	; 右超声波
ORB
OUT    Y10006	; 右超声波启动
LD     M1001	; 自动运行中
ANI    HM1	; on，测试，off有料运行
LDI    HM30	; off手动 ON自动
AND    M9960
ORB
LD     Y10007	; 上线对接信号
AND    HM30	; off手动 ON自动
ORB
LDI    M24	; 来料感应
ANI    T107
ANI    SM1000
ORI    HM30	; off手动 ON自动
ANB
OUT    Y10007	; 上线对接信号
LD     Y10007	; 上线对接信号
TMR    T107 HD9950 K1
LDI    HM31	; off使能
AND    SM1
OUT    Y10010	; 伺服使能
LD     M13	; 报警清除
OUT    Y10011	; 伺服报警清除
LD     M506	; 左双夹耳气缸
ANI    M406	; 气缸6/手动
LDI    M506	; 左双夹耳气缸
AND    M406	; 气缸6/手动
ORB
OUT    Y10012	; 左双夹
LD     M504	; 左压耳带气缸
ANI    M404	; 气缸4/手动
LD     M404	; 气缸4/手动
ANI    M504	; 左压耳带气缸
ORB
OUT    Y10013	; 左压夹耳带

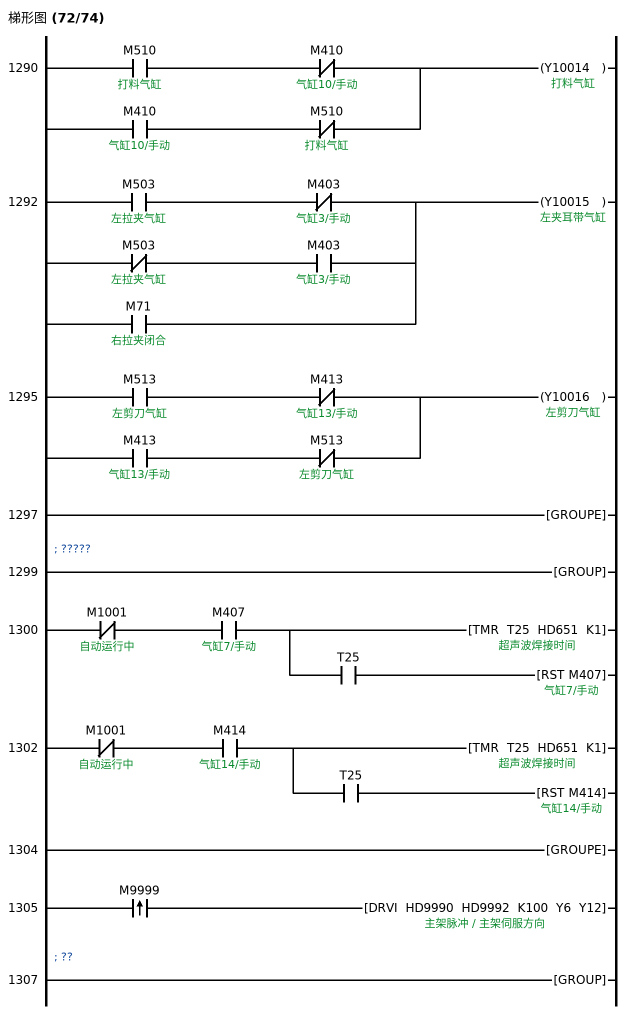
LD     M510	; 打料气缸
ANI    M410	; 气缸10/手动
LD     M410	; 气缸10/手动
ANI    M510	; 打料气缸
ORB
OUT    Y10014	; 打料气缸
LD     M503	; 左拉夹气缸
ANI    M403	; 气缸3/手动
LDI    M503	; 左拉夹气缸
AND    M403	; 气缸3/手动
ORB
OR     M71	; 右拉夹闭合
OUT    Y10015	; 左夹耳带气缸
LD     M513	; 左剪刀气缸
ANI    M413	; 气缸13/手动
LD     M413	; 气缸13/手动
ANI    M513	; 左剪刀气缸
ORB
OUT    Y10016	; 左剪刀气缸
GROUPE
; ?????
GROUP
LDI    M1001	; 自动运行中
AND    M407	; 气缸7/手动
TMR    T25 HD651 K1	; 超声波焊接时间
AND    T25
RST    M407	; 气缸7/手动
LDI    M1001	; 自动运行中
AND    M414	; 气缸14/手动
TMR    T25 HD651 K1	; 超声波焊接时间
AND    T25
RST    M414	; 气缸14/手动
GROUPE
LDP    M9999
DRVI   HD9990 HD9992 K100 Y6 Y12	; 主架脉冲 / 主架伺服方向
; ??
GROUP

